// TIA Portal V20 export
DATA_BLOCK "Station_MOVIKIT"   // DB23
{ S7_Optimized_Access := 'TRUE' }
// stored: MemoryReserve 100
   VAR
      MStNONE_PI : "SEW_MOVIKIT_VelocityDrive_STATUS_V2.1";
      MStNONE_PO : "SEW_MOVIKIT_VelocityDrive_SETPOINTS_V2.1";
      MSt1_PI : "SEW_MOVIKIT_VelocityDrive_STATUS_V2.1";
      MSt1_PO : "SEW_MOVIKIT_VelocityDrive_SETPOINTS_V2.1";
      MSt1a_PI : "SEW_MOVIKIT_VelocityDrive_STATUS_V2.1";
      MSt1a_PO : "SEW_MOVIKIT_VelocityDrive_SETPOINTS_V2.1";
      MSt4a_PI : "SEW_MOVIKIT_VelocityDrive_STATUS_V2.1";
      MSt4a_PO : "SEW_MOVIKIT_VelocityDrive_SETPOINTS_V2.1";
      MSt4b_PI : "SEW_MOVIKIT_VelocityDrive_STATUS_V2.1";
      MSt4b_PO : "SEW_MOVIKIT_VelocityDrive_SETPOINTS_V2.1";
      MSt5_PI : "SEW_MOVIKIT_VelocityDrive_STATUS_V2.1";
      MSt5_PO : "SEW_MOVIKIT_VelocityDrive_SETPOINTS_V2.1";
      MSt6a_PI : "SEW_MOVIKIT_VelocityDrive_STATUS_V2.1";
      MSt6a_PO : "SEW_MOVIKIT_VelocityDrive_SETPOINTS_V2.1";
      MSt6b_PI : "SEW_MOVIKIT_VelocityDrive_STATUS_V2.1";
      MSt6b_PO : "SEW_MOVIKIT_VelocityDrive_SETPOINTS_V2.1";
      MSt7_PI : "SEW_MOVIKIT_VelocityDrive_STATUS_V2.1";
      MSt7_PO : "SEW_MOVIKIT_VelocityDrive_SETPOINTS_V2.1";
      MSt8_PI : "SEW_MOVIKIT_VelocityDrive_STATUS_V2.1";
      MSt8_PO : "SEW_MOVIKIT_VelocityDrive_SETPOINTS_V2.1";
      MSt9a_PI : "SEW_MOVIKIT_VelocityDrive_STATUS_V2.1";
      MSt9a_PO : "SEW_MOVIKIT_VelocityDrive_SETPOINTS_V2.1";
      MSt9b_PI : "SEW_MOVIKIT_VelocityDrive_STATUS_V2.1";
      MSt9b_PO : "SEW_MOVIKIT_VelocityDrive_SETPOINTS_V2.1";
      MSt10_PI : "SEW_MOVIKIT_VelocityDrive_STATUS_V2.1";
      MSt10_PO : "SEW_MOVIKIT_VelocityDrive_SETPOINTS_V2.1";
      MSt11_PI : "SEW_MOVIKIT_VelocityDrive_STATUS_V2.1";
      MSt11_PO : "SEW_MOVIKIT_VelocityDrive_SETPOINTS_V2.1";
      MSt12a_PI : "SEW_MOVIKIT_VelocityDrive_STATUS_V2.1";
      MSt12a_PO : "SEW_MOVIKIT_VelocityDrive_SETPOINTS_V2.1";
      MSt12b_PI : "SEW_MOVIKIT_VelocityDrive_STATUS_V2.1";
      MSt12b_PO : "SEW_MOVIKIT_VelocityDrive_SETPOINTS_V2.1";
      MSt13_PI : "SEW_MOVIKIT_VelocityDrive_STATUS_V2.1";
      MSt13_PO : "SEW_MOVIKIT_VelocityDrive_SETPOINTS_V2.1";
      MSt14_PI : "SEW_MOVIKIT_VelocityDrive_STATUS_V2.1";
      MSt14_PO : "SEW_MOVIKIT_VelocityDrive_SETPOINTS_V2.1";
      MSt17_PI : "SEW_MOVIKIT_VelocityDrive_STATUS_V2.1";
      MSt17_PO : "SEW_MOVIKIT_VelocityDrive_SETPOINTS_V2.1";
      MSt18_PI : "SEW_MOVIKIT_VelocityDrive_STATUS_V2.1";
      MSt18_PO : "SEW_MOVIKIT_VelocityDrive_SETPOINTS_V2.1";
      MSt19a_PI : "SEW_MOVIKIT_VelocityDrive_STATUS_V2.1";
      MSt19a_PO : "SEW_MOVIKIT_VelocityDrive_SETPOINTS_V2.1";
      MSt19b_PI : "SEW_MOVIKIT_VelocityDrive_STATUS_V2.1";
      MSt19b_PO : "SEW_MOVIKIT_VelocityDrive_SETPOINTS_V2.1";
      MSt20_PI : "SEW_MOVIKIT_VelocityDrive_STATUS_V2.1";
      MSt20_PO : "SEW_MOVIKIT_VelocityDrive_SETPOINTS_V2.1";
      MSt21_PI : "SEW_MOVIKIT_VelocityDrive_STATUS_V2.1";
      MSt21_PO : "SEW_MOVIKIT_VelocityDrive_SETPOINTS_V2.1";
      MSt22a_PI : "SEW_MOVIKIT_VelocityDrive_STATUS_V2.1";
      MSt22a_PO : "SEW_MOVIKIT_VelocityDrive_SETPOINTS_V2.1";
      MSt22b_PI : "SEW_MOVIKIT_VelocityDrive_STATUS_V2.1";
      MSt22b_PO : "SEW_MOVIKIT_VelocityDrive_SETPOINTS_V2.1";
      MSt23a_PI : "SEW_MOVIKIT_VelocityDrive_STATUS_V2.1";
      MSt23a_PO : "SEW_MOVIKIT_VelocityDrive_SETPOINTS_V2.1";
      MSt23b_PI : "SEW_MOVIKIT_VelocityDrive_STATUS_V2.1";
      MSt23b_PO : "SEW_MOVIKIT_VelocityDrive_SETPOINTS_V2.1";
      MSt24a_PI : "SEW_MOVIKIT_VelocityDrive_STATUS_V2.1";
      MSt24a_PO : "SEW_MOVIKIT_VelocityDrive_SETPOINTS_V2.1";
      MSt24b_PI : "SEW_MOVIKIT_VelocityDrive_STATUS_V2.1";
      MSt24b_PO : "SEW_MOVIKIT_VelocityDrive_SETPOINTS_V2.1";
      MSt25a_PI : "SEW_MOVIKIT_VelocityDrive_STATUS_V2.1";
      MSt25a_PO : "SEW_MOVIKIT_VelocityDrive_SETPOINTS_V2.1";
      MSt25b_PI : "SEW_MOVIKIT_VelocityDrive_STATUS_V2.1";
      MSt25b_PO : "SEW_MOVIKIT_VelocityDrive_SETPOINTS_V2.1";
      MSt26_PI : "SEW_MOVIKIT_VelocityDrive_STATUS_V2.1";
      MSt26_PO : "SEW_MOVIKIT_VelocityDrive_SETPOINTS_V2.1";
      MSt27a_PI : "SEW_MOVIKIT_VelocityDrive_STATUS_V2.1";
      MSt27a_PO : "SEW_MOVIKIT_VelocityDrive_SETPOINTS_V2.1";
      MSt27b_PI : "SEW_MOVIKIT_VelocityDrive_STATUS_V2.1";
      MSt27b_PO : "SEW_MOVIKIT_VelocityDrive_SETPOINTS_V2.1";
      MSt28_PI : "SEW_MOVIKIT_VelocityDrive_STATUS_V2.1";
      MSt28_PO : "SEW_MOVIKIT_VelocityDrive_SETPOINTS_V2.1";
      MSt29_PI : "SEW_MOVIKIT_VelocityDrive_STATUS_V2.1";
      MSt29_PO : "SEW_MOVIKIT_VelocityDrive_SETPOINTS_V2.1";
      MSt30b_PI : "SEW_MOVIKIT_VelocityDrive_STATUS_V2.1";
      MSt30b_PO : "SEW_MOVIKIT_VelocityDrive_SETPOINTS_V2.1";
      MSt30a_PI : "SEW_MOVIKIT_VelocityDrive_STATUS_V2.1";
      MSt30a_PO : "SEW_MOVIKIT_VelocityDrive_SETPOINTS_V2.1";
      MSt31_PI : "SEW_MOVIKIT_VelocityDrive_STATUS_V2.1";
      MSt31_PO : "SEW_MOVIKIT_VelocityDrive_SETPOINTS_V2.1";
      MSt32_PI : "SEW_MOVIKIT_VelocityDrive_STATUS_V2.1";
      MSt32_PO : "SEW_MOVIKIT_VelocityDrive_SETPOINTS_V2.1";
      MSt33a_PI : "SEW_MOVIKIT_VelocityDrive_STATUS_V2.1";
      MSt33a_PO : "SEW_MOVIKIT_VelocityDrive_SETPOINTS_V2.1";
      MSt33b_PI : "SEW_MOVIKIT_VelocityDrive_STATUS_V2.1";
      MSt33b_PO : "SEW_MOVIKIT_VelocityDrive_SETPOINTS_V2.1";
      MSt34_PI : "SEW_MOVIKIT_VelocityDrive_STATUS_V2.1";
      MSt34_PO : "SEW_MOVIKIT_VelocityDrive_SETPOINTS_V2.1";
      MSt35_PI : "SEW_MOVIKIT_VelocityDrive_STATUS_V2.1";
      MSt35_PO : "SEW_MOVIKIT_VelocityDrive_SETPOINTS_V2.1";
      MSt36a_PI : "SEW_MOVIKIT_VelocityDrive_STATUS_V2.1";
      MSt36a_PO : "SEW_MOVIKIT_VelocityDrive_SETPOINTS_V2.1";
      MSt36b_PI : "SEW_MOVIKIT_VelocityDrive_STATUS_V2.1";
      MSt36b_PO : "SEW_MOVIKIT_VelocityDrive_SETPOINTS_V2.1";
      MSt37_PI : "SEW_MOVIKIT_VelocityDrive_STATUS_V2.1";
      MSt37_PO : "SEW_MOVIKIT_VelocityDrive_SETPOINTS_V2.1";
      MSt38_PI : "SEW_MOVIKIT_VelocityDrive_STATUS_V2.1";
      MSt38_PO : "SEW_MOVIKIT_VelocityDrive_SETPOINTS_V2.1";
   END_VAR
BEGIN
   MStNONE_PI.x_Bit_0_Ready := 1;
END_DATA_BLOCK
